{attribute 'qualified_only'}
{attribute 'strict'}
{attribute 'to_string'}
TYPE E_FilterType :
(	
	Disabled := 0,
	PTn,
	MovingAverage
);
END_TYPE

(* stored: Version 1.1.0.1, ProductVersion 3.1.4026.17
   DUT E_FilterType: Id {02893b45-df21-4124-bf38-e1ffc2721c82} *)
